# EPICS substitutions: ek9000App/Db/EL3208.substitutions
file EL3208.template
{ 	pattern
	{
		TERMINAL,

	}
	{
	}
}

	}
	{
	}
}

	}
	{
	}
}

	}
	{
	}
}

	}
	{
	}
}

	}
	{
	}
}

	}
	{
	}
}

	}
	{
	}
}
